Universal Robots PolyScope program: tangram.urp

Program tangram (installation=comm directory=/programs/usbdisk/RobotControl createdIn=5.14.5 lastSavedIn=5.14.5 robotSerialNumber=20225501312)
Calibrated DH parameters: a=[0.000177, -0.405867, -0.359302, -0.000009, 0.00008, 0]; d=[0.162556, -59.259033, 22.634856, 36.757695, 0.099775, 0.099535]; alpha=[1.570983, 0.00214, 0.004319, 1.570342, -1.569638, 0]; deltaTheta=[0, -0.302866, 6.171309, 0.414749, 0.000002, -0.000001]
InitVariablesNode variables(variable(name=PLOC_Ref, expression=[0.000000,-1.570800,-1.570800,-1.745330,1.570800,1.570800]), variable(name=PLOC_clear, expression=p[0,0,0,0,0,0]), variable(name=PLOC_pick, expression=p[0,0,0,0,0,0]), variable(name=PLOC_prepick, expression=[0,0,0,0,0,0]), variable(name=PLOC_total_33, expression=0), variable(name=PLOC_total_34, expression=0), variable(name=n_shapes, expression=0))
BeforeStart
  URCap Gripper Activate (Robotiq_Grippers, Robotiq Inc.) dataModel(ResetAndActivateKey=false)
  URCap Gripper (Robotiq_Grippers, Robotiq Inc.) dataModel(position=0.0, force=100.0, speed=100.0, positionInDouble=0.0, forceInDouble=100.0, speedInDouble=100.0, slaveIds=[9], blocking=true, robotCompliant=false)
  l := make_list(42, 0)
  open_socket := socket_open("192.168.65.161", 8888, "ur5e_pc")
  Loop While (checkContinuously=false) expression=open_socket≟ False
    open_socket := socket_open("192.168.65.161", 8888, "ur5e_pc")
  placing_offset := p[0,0,-0.02,0,0,0]
  rpy_base := rotvec2rpy([2.225, -2.208, 0])
  orient := [0,0,0]
  recv_i := 0
  i := 0
  str_ack := ""
  is_receiving := False
  SuppressedNode
    Loop While (checkContinuously=false) expression=is_receiving≟ False
      socket_data := socket_read_ascii_float(6,"ur5e_pc")
      If socket_data[0]≠0
        is_receiving := True
      Wait Sleep waitTime=0.01
  Loop Counting (count=7) loopVariable(name=Loop_2)
    Loop While (checkContinuously=false) expression=str_ack≠"ACK"
      str_ack := socket_read_string("ur5e_pc")
      Wait Sleep waitTime=0.01
    socket_data := socket_read_ascii_float(6,"ur5e_pc")
    Loop While (checkContinuously=false) expression=socket_data[0]≠6
      socket_data := socket_read_ascii_float(6,"ur5e_pc")
      Wait Sleep waitTime=0.1
    Loop While (checkContinuously=false) expression=recv_i<6
      Script: l[i]=socket_data[recv_i+1]
      i := i+1
      recv_i := recv_i+1
      SuppressedNode
        square := [socket_data.slice(1, 6)]
    SuppressedNode
      l := l.append([socket_data[1], socket_data[2], socket_data[3],socket_data[4],socket_data[5],socket_data[6], socket_data[7]])
    SuppressedNode
      Script: l.append([socket_data[1], socket_data[2], socket_data[3], socket_data[4], socket_data[5], socket_data[6]])
    recv_i := 0
    ack_send := socket_send_string("ACK","ur5e_pc")
    Loop While (checkContinuously=false) expression=ack_send≟ False
      ack_send := socket_send_string("ACK","ur5e_pc")
      Wait Sleep waitTime=0.01
  SuppressedNode
    Popup Warning (haltProgram=false message=debug inputType=Text)
  SuppressedNode
    l := socket_data
  triangle_mid := p[l[0],l[1],l[2],l[3],l[4],l[5]]
  triangle_s1 := p[l[6],l[7],l[8],l[9],l[10],l[11]]
  triangle_s2 := p[l[12],l[13],l[14],l[15],l[16],l[17]]
  triangle_big1 := p[l[18],l[19],l[20],l[21],l[22],l[23]]
  triangle_big2 := p[l[24],l[25],l[26],l[27],l[28],l[29]]
  square := p[l[30],l[31],l[32],l[33],l[34],l[35]]
  parallelogram := p[l[36],l[37],l[38],l[39],l[40],l[41]]
  cam_offset := p[0.02,0,-0.025,0,0,1.570]
  i := 0
  n_shapes := 7   [initializeExpression=0]
  trgsm_n := 1
  trgbig_n := 1
  MoveJ speed 60 deg/s, acceleration 80 deg/s^2 (useActiveTCP=false) tcp=TCPfingers; feature=Base
    Waypoint Start: motionParameters(blendRadius=0.01); TCP in base x=456.475 y=-121.214 z=87.765 mm, rx=2.225 ry=-2.2083 rz=-0.0179 rad; joints [1.47, -95.414, -120.916, -54.463, 90.369, 1.109] deg; TCP offset x=0 y=0 z=165 mm, rx=0 ry=0 rz=0 rad
Robot Program (runOnlyOnce=true)
  Loop While (checkContinuously=false) expression=i < n_shapes
    SuppressedNode
      Popup Message (haltProgram=false message=i inputType=Text)
    URCap PLOC2D (PART LOCALIZATION WITH SICK PLOC2D, SICK AG - Developed by Nimalendiran Kailasanathan) dataModel(Z_OFFSET=0.0, IS_ABOVE_BIN_SET_KEY=true, SELECTED_JOBS=1 2 3 4 5 , LOCALIZATION_TIMEOUT=10, IP_ADDRESS_LIST_OF=[192.168.65.216], IS_PICK_ALL_PARTS_SELECTED=1, SELECTED_IP_ADDRESS=192.168.65.216, SELECTED_ALIGNMENT_NAME=sick_cam, Variable(key=PLOC_REF_POSE_KEY, variable(name=PLOC_Ref, initializeExpression=[0.000000,-1.570800,-1.570800,-1.745330,1.570800,1.570800])), Variable(key=PLOC_PRE_PICK_POSE, variable(name=PLOC_prepick, initializeExpression=[0,0,0,0,0,0])), Variable(key=PLOC_PICK_POSE, variable(name=PLOC_pick, initializeExpression=p[0,0,0,0,0,0])), Variable(key=PLOC_CLEAR_POSE_KEY, variable(name=PLOC_clear, initializeExpression=p[0,0,0,0,0,0])), TCP(key=selected-tcp name=TCPfingers), JointPositions(key=JOINT_REF_ANGLES, JointPosition(key=[1], Angle(key=pos value=0.64209 unit=RAD)), JointPosition(key=[2], Angle(key=pos value=-1.79064 unit=RAD)), JointPosition(key=[3], Angle(key=pos value=-2.2028 unit=RAD)), JointPosition(key=[4], Angle(key=pos value=-0.73302 unit=RAD)), JointPosition(key=[5], Angle(key=pos value=1.57761 unit=RAD)), JointPosition(key=[6], Angle(key=pos value=0.62786 unit=RAD))), Variable(key=TOTAL_VAR, variable(name=PLOC_total_33, initializeExpression=0)), Variable(key=NUMBER_OF_MATCHES_VAR, variable(name=PLOC_total_34, initializeExpression=0)), Pose(key=SELECTED_ALIGNMENT_POSE, Position(key=posePosition, Length(key=X value=0.43363 unit=M), Length(key=Y value=0.17376 unit=M), Length(key=Z value=0.05179 unit=M)), Rotation(key=poseRotation, Angle(key=RX value=2.21728 unit=RAD), Angle(key=RY value=2.21672 unit=RAD), Angle(key=RZ value=-0.02909 unit=RAD))))
      Folder Folder
        Folder Pick and Place
          Folder Start
            'Set start position and open gripper'
            MoveJ speed 60 deg/s, acceleration 80 deg/s^2 (useActiveTCP=false) tcp=TCPfingers; feature=Base
              Waypoint Start: motionParameters(blendRadius=0.01); TCP in base x=456.475 y=-121.214 z=87.765 mm, rx=2.225 ry=-2.2083 rz=-0.0179 rad; joints [1.47, -95.414, -120.916, -54.463, 90.369, 1.109] deg
          SuppressedNode
            n_shapes := PLOC_total_1
          SuppressedNode
            Halt
          Folder Approach
            MoveJ speed 60 deg/s, acceleration 80 deg/s^2 (useActiveTCP=false) tcp=TCPfingers; feature=Base
              Waypoint Variable (Variable): motionParameters(blendRadius=0.01); variable=PLOC_prepick
          Folder Pick
            PLOC_pick := pose_add(PLOC_pick,cam_offset)
            MoveL speed 250 mm/s, acceleration 1200 mm/s^2 (useActiveTCP=false) tcp=TCPfingers; feature=Base
              Waypoint Variable (Variable): variable=PLOC_pick
              SuppressedNode
                Halt
            URCap Gripper (Robotiq_Grippers, Robotiq Inc.) dataModel(position=100.0, force=100.0, speed=100.0, positionInDouble=100.0, forceInDouble=100.0, speedInDouble=100.0, slaveIds=[9], blocking=true, robotCompliant=false)
          Folder Clear
            'Close gripper'
            MoveL speed 250 mm/s, acceleration 1200 mm/s^2 (useActiveTCP=false) tcp=TCPfingers; feature=Base
              Waypoint Variable (Variable): motionParameters(blendRadius=0.01); variable=PLOC_clear
          Folder Place
            'Set drop position and open gripper'
            shitrobot := PLOC2D_JOB_ID
            SuppressedNode
              Popup Message (haltProgram=false inputType=Variable) variable=shitrobot
            If shitrobot ≟ 1
              orient := rpy2rotvec(rpy_base+[0,0,triangle_mid[5]])
              SuppressedNode
                triangle_mid := pose_add(triangle_mid, p[0,0,0,orient[0], orient[1], orient[2]])
              triangle_mid := p[triangle_mid[0], triangle_mid[1], triangle_mid[2],orient[0], orient[1], orient[2]]
              debug1 := rotvec2rpy([triangle_mid[5], triangle_mid[4], triangle_mid[5]])
              MoveJ speed 60 deg/s, acceleration 80 deg/s^2 (useActiveTCP=false) tcp=TCPfingers; feature=Base
                Waypoint Variable (Variable): variable=triangle_mid
                triangle_mid := pose_add(triangle_mid, placing_offset)
              MoveJ speed 60 deg/s, acceleration 80 deg/s^2 (useActiveTCP=false) tcp=TCPfingers; feature=Base
                Waypoint Variable (Variable): variable=triangle_mid
                URCap Gripper (Robotiq_Grippers, Robotiq Inc.) dataModel(position=0.0, force=100.0, speed=100.0, positionInDouble=0.0, forceInDouble=100.0, speedInDouble=100.0, slaveIds=[9], blocking=true, robotCompliant=false)
            ElseIf shitrobot ≟ 2
              If trgsm_n≟1
                orient := rpy2rotvec(rpy_base+[0,0,triangle_s1[5]])
                triangle_s1 := pose_add(triangle_s1, p[0,0,0,orient[0], orient[1], orient[2]])
                MoveJ speed 60 deg/s, acceleration 80 deg/s^2 (useActiveTCP=true) feature=Base
                  Waypoint Variable (Variable): variable=triangle_s1
                  triangle_s1 := pose_add(triangle_s1, placing_offset)
                MoveJ speed 60 deg/s, acceleration 80 deg/s^2 (useActiveTCP=true) feature=Base
                  Waypoint Variable (Variable): variable=triangle_s1
                  URCap Gripper (Robotiq_Grippers, Robotiq Inc.) dataModel(position=0.0, force=100.0, speed=100.0, positionInDouble=0.0, forceInDouble=100.0, speedInDouble=100.0, slaveIds=[9], blocking=true, robotCompliant=false)
                trgsm_n := trgsm_n+1
              Else 
                orient := rpy2rotvec(rpy_base+[0,0,triangle_s2[5]])
                triangle_s2 := pose_add(triangle_s2, p[0,0,0,orient[0], orient[1], orient[2]])
                MoveJ speed 60 deg/s, acceleration 80 deg/s^2 (useActiveTCP=true) feature=Base
                  Waypoint Variable (Variable): variable=triangle_s2
                  triangle_s2 := pose_add(triangle_s1, placing_offset)
                MoveJ speed 60 deg/s, acceleration 80 deg/s^2 (useActiveTCP=true) feature=Base
                  Waypoint Variable (Variable): variable=triangle_s2
                  URCap Gripper (Robotiq_Grippers, Robotiq Inc.) dataModel(position=0.0, force=100.0, speed=100.0, positionInDouble=0.0, forceInDouble=100.0, speedInDouble=100.0, slaveIds=[9], blocking=true, robotCompliant=false)
            ElseIf shitrobot ≟ 3
              SuppressedNode
                MoveJ speed 60 deg/s, acceleration 80 deg/s^2 (useActiveTCP=true) feature=Base
                  Waypoint Variable (Variable): variable=triangle_big1
                  triangle_big1 := pose_add(triangle_big1, placing_offset)
              If trgbig_n≟1
                orient := rpy2rotvec(rpy_base+[0,0,triangle_big1[5]])
                triangle_big1 := pose_add(triangle_big1, p[0,0,0,orient[0], orient[1], orient[2]])
                MoveJ speed 60 deg/s, acceleration 80 deg/s^2 (useActiveTCP=true) feature=Base
                  Waypoint Variable (Variable): variable=triangle_big1
                  triangle_big1 := pose_add(triangle_big1, placing_offset)
                MoveJ speed 60 deg/s, acceleration 80 deg/s^2 (useActiveTCP=true) feature=Base
                  Waypoint Variable (Variable): variable=triangle_big1
                  URCap Gripper (Robotiq_Grippers, Robotiq Inc.) dataModel(position=0.0, force=100.0, speed=100.0, positionInDouble=0.0, forceInDouble=100.0, speedInDouble=100.0, slaveIds=[9], blocking=true, robotCompliant=false)
                trgbig_n := trgbig_n+1
              Else 
                orient := rpy2rotvec(rpy_base+[0,0,triangle_big2[5]])
                triangle_big2 := pose_add(triangle_big2, p[0,0,0,orient[0], orient[1], orient[2]])
                MoveJ speed 60 deg/s, acceleration 80 deg/s^2 (useActiveTCP=true) feature=Base
                  Waypoint Variable (Variable): variable=triangle_big2
                  triangle_big2 := pose_add(triangle_big2, placing_offset)
                MoveJ speed 60 deg/s, acceleration 80 deg/s^2 (useActiveTCP=true) feature=Base
                  Waypoint Variable (Variable): variable=triangle_big2
                  URCap Gripper (Robotiq_Grippers, Robotiq Inc.) dataModel(position=0.0, force=100.0, speed=100.0, positionInDouble=0.0, forceInDouble=100.0, speedInDouble=100.0, slaveIds=[9], blocking=true, robotCompliant=false)
              MoveJ speed 60 deg/s, acceleration 80 deg/s^2 (useActiveTCP=true) feature=Base
                Waypoint Variable (Variable): variable=triangle_big1
                URCap Gripper (Robotiq_Grippers, Robotiq Inc.) dataModel(position=0.0, force=100.0, speed=100.0, positionInDouble=0.0, forceInDouble=100.0, speedInDouble=100.0, slaveIds=[9], blocking=true, robotCompliant=false)
            ElseIf shitrobot ≟ 4
              orient := rpy2rotvec(rpy_base+[0,0,square[5]])
              square := pose_add(square, p[0,0,0,orient[0], orient[1], orient[2]])
              MoveJ speed 60 deg/s, acceleration 80 deg/s^2 (useActiveTCP=false) tcp=TCPfingers; feature=Base
                Waypoint Variable (Variable): variable=square
                square := pose_add(square, placing_offset)
              MoveJ speed 60 deg/s, acceleration 80 deg/s^2 (useActiveTCP=true) feature=Base
                Waypoint Variable (Variable): variable=square
                URCap Gripper (Robotiq_Grippers, Robotiq Inc.) dataModel(position=0.0, force=100.0, speed=100.0, positionInDouble=0.0, forceInDouble=100.0, speedInDouble=100.0, slaveIds=[9], blocking=true, robotCompliant=false)
            ElseIf shitrobot ≟ 5
              orient := rpy2rotvec(rpy_base+[0,0,parallelogram[5]])
              parallelogram := pose_add(parallelogram, p[0,0,0,orient[0], orient[1], orient[2]])
              MoveJ speed 60 deg/s, acceleration 80 deg/s^2 (useActiveTCP=false) tcp=TCPfingers; feature=Base
                Waypoint Variable (Variable): variable=parallelogram
                parallelogram := pose_add(parallelogram, placing_offset)
              MoveJ speed 60 deg/s, acceleration 80 deg/s^2 (useActiveTCP=true) feature=Base
                Waypoint Variable (Variable): variable=parallelogram
                URCap Gripper (Robotiq_Grippers, Robotiq Inc.) dataModel(position=0.0, force=100.0, speed=100.0, positionInDouble=0.0, forceInDouble=100.0, speedInDouble=100.0, slaveIds=[9], blocking=true, robotCompliant=false)
    i := i+1
  MoveJ speed 60 deg/s, acceleration 80 deg/s^2 (useActiveTCP=false) tcp=TCPfingers; feature=Base
    Waypoint Start: motionParameters(blendRadius=0.01); TCP in base x=456.475 y=-121.214 z=87.765 mm, rx=2.225 ry=-2.2083 rz=-0.0179 rad; joints [1.47, -95.414, -120.916, -54.463, 90.369, 1.109] deg
